TYPE UpdaterEntry :
STRUCT
	TypeID	: BYTE;
	Version	: BYTE;
	Updater	: ITF_Updater;
END_STRUCT
END_TYPE

(* stored: Version 1.1.0.1
   DUT UpdaterEntry: Id {929be010-92ad-4ce6-9437-b7a7b3639152} *)
